// TwinCAT 3 PLC project Simulation
// ProgramVersion: 3.1.4023.0
// libraries:
//   Tc2_ControllerToolbox, * (Beckhoff Automation GmbH)
//   Tc2_Standard, * (Beckhoff Automation GmbH)
//   Tc2_System, * (Beckhoff Automation GmbH)
//   Tc2_TempController, * (Beckhoff Automation GmbH)
//   Tc3_Module, * (Beckhoff Automation GmbH)
// project tree:
//   / PlcTask.TcTTO
//   POUs/ FB_Process.TcPOU, MAIN.TcPOU
// (motion and I/O tree: see PLC project plc01)
// real-time tasks:
//   TASK PlcTask: cycle T#10ms, priority 20, ADS port 350
//   TASK PlcTask1: cycle T#10ms, priority 21, ADS port 351
// variable links:
//   PLC01 Instance <-> Simulation/Simulation Instance
//     PlcTask Inputs/MAIN.currTemp <-> PlcTask Outputs/MAIN.actualTemp
//     PlcTask Outputs/MAIN.fyAnalogOutput <-> PlcTask Inputs/MAIN.tempCmd

CONFIGURATION Simulation
    RESOURCE PLC ON TwinCAT3
        TASK PlcTask(INTERVAL := T#10ms, PRIORITY := 21);
        PROGRAM MAIN WITH PlcTask : MAIN;
    END_RESOURCE
END_CONFIGURATION

// ---- POUs/MAIN.TcPOU
PROGRAM MAIN
VAR
	temperatureSimul:FB_Process;
	tempCmd AT %I*:LREAL;
	actualTemp AT %Q*:LREAL;
END_VAR
VAR CONSTANT
	taskCycletime:TIME:=T#10MS;
	bNoiseEnable:BOOL:=TRUE;
END_VAR

temperatureSimul(fY:= tempCmd, tTa:=taskCycletime , bNoise:= bNoiseEnable, fX=>actualTemp);

END_PROGRAM

// ---- POUs/FB_Process.TcPOU
FUNCTION_BLOCK FB_Process

VAR_INPUT
	fY		:	LREAL;
	tTa		:	TIME;
	bNoise	:	BOOL;
END_VAR

VAR_OUTPUT
	fX		:	LREAL;
END_VAR

VAR
	(* Processparameters *)
	tT11		:	TIME	:= t#5s;
	tT12		:	TIME	:= t#25s;

	(* process *)
	fbProcessPart1	:	FB_CTRL_PT1;
	fbProcessPart2	:	FB_CTRL_PT1;
	fbNoise			:	FB_CTRL_NOISE_GENERATOR;

	stProcessPart1	:	ST_CTRL_PT1_PARAMS;
	stProcessPart2	:	ST_CTRL_PT1_PARAMS;
	stNoise			:	ST_CTRL_NOISE_GENERATOR_PARAMS;
	
END_VAR

(* init structures *)
stProcessPart1.fKp := 1.0;
stProcessPart1.tCtrlCycleTime := tTa;
stProcessPart1.tT1 := tT11;
stProcessPart1.tTaskCycleTime := tTa;

stProcessPart2.fKp := 1.0;
stProcessPart2.tCtrlCycleTime := tTa;
stProcessPart2.tT1 := tT12;
stProcessPart2.tTaskCycleTime := tTa;

stNoise.fAmplitude := 1.0;
stNoise.tCtrlCycleTime := tTa;
stNoise.tTaskCycleTime := tTa;

(* calculate and simulate process *)
fbProcessPart1(
				fIn:= fY,
				fManSyncValue:= 0.0,
				bSync:= FALSE,
				eMode:= eCTRL_MODE_ACTIVE,
				bHold:= FALSE,
				stParams:= stProcessPart1);

fbProcessPart2(
				fIn:= fbProcessPart1.fOut,
				fManSyncValue:= 0.0,
				bSync:= FALSE,
				eMode:= eCTRL_MODE_ACTIVE,
				bHold:= FALSE,
				stParams:= stProcessPart2);

fbNoise(
		fManSyncValue:= 0.0,
		eMode:= eCTRL_MODE_ACTIVE,
		stParams:= stNoise);

IF bNoise THEN
	fX := fbProcessPart2.fOut + 0.01*fbNoise.fOut;
ELSE
	fX := fbProcessPart2.fOut;
END_IF;

END_FUNCTION_BLOCK
